(* Logix 5000 project; controller AlarmsWithModbus vendor 1 type 14 code 164 rev 38.11; software revision 38.01 *)

TASK MainTask (continuous, watchdog 500 ms) : MainProgram

MODULES
   Local : vendor 1 type 14 code 164 (ICP 4, rev 38.11)
END_MODULES

VAR_GLOBAL   (* controller tags *)
   Alarm1 : BOOL;
   Alarm2 : BOOL;
   Alarm3 : BOOL;
END_VAR

PROGRAM MainProgram   (* main routine MainRoutine *)

ROUTINE MainRoutine   (* ladder *)
END_ROUTINE
END_PROGRAM
